(* CoDeSys 2.3 export: ST_MQTTTELEGRAM.EXP *)

(* Data type *)
TYPE ST_MqttTelegram :
STRUCT
	arMqttData 	: ARRAY[0..544] OF BYTE;
	nDataLength	: UDINT := 0;
END_STRUCT
END_TYPE
